Yaskawa INFORM job: R1_W39(90,0)R2.JBI

/JOB
//NAME R1_W39(90,0)R2
///FOLDERNAME KRIS-SCIANA
//POS
///NPOS 43,43,0,0,0,0
///TOOL 0
///POSTYPE PULSE
///PULSE
C00000=-48919,8763,-78145,-33912,86192,59629
C00001=-76192,74539,-3713,-7584,90498,58184
C00002=-85002,92103,26363,-6620,109146,2540
C00003=-82989,104273,47097,-9079,108858,2634
C00004=-80348,97044,37326,-14355,108478,2463
C00005=-80254,95353,36923,-14306,107890,2566
C00006=-81479,107840,53058,-15936,109964,1832
C00007=-88415,93116,33475,-16240,113040,-1015
C00008=-84401,99025,43999,-26670,113361,-1779
C00009=-80535,97927,39068,-19437,112108,13102
C00010=-80533,100008,38267,-19688,113585,12840
C00011=-95804,89991,27481,9151,105821,-39381
C00012=-93260,116784,65555,9230,104296,-50461
C00013=-88855,89918,29422,-607,100748,-50698
C00014=-93687,111856,59478,9313,105536,-50507
C00015=-89184,93974,34704,-472,103135,-51673
C00016=-95648,113896,64634,12639,107588,-50809
C00017=-91220,113921,60892,3414,106966,-50938
C00018=-94799,78029,20878,7231,106457,-51217
C00019=-94338,106165,52191,9314,107335,-50796
C00020=-97825,95185,41124,15323,107662,-50686
C00021=-97701,80312,23794,13413,106555,-50896
C00022=-97503,99676,37498,14313,114598,-56335
C00023=-97503,101438,37062,14468,115737,-56186
C00024=-130465,99741,46634,38839,105281,12352
C00025=-128682,100738,50844,38236,102897,12201
C00026=-125742,101757,54133,37646,100487,12538
C00027=-117769,55117,-4342,7008,90476,33925
C00028=-118319,57270,-3229,7217,90935,33791
C00029=-127381,86615,37635,37885,96810,10695
C00030=-119102,89171,33145,15718,101015,10229
C00031=-114648,83746,25609,1808,100380,9031
C00032=-114353,83732,25539,225,100330,11365
C00033=-114685,81630,17220,455,104304,11368
C00034=-111532,73347,14192,-9053,100688,13279
C00035=-111918,74812,15995,-7480,100020,12650
C00036=-113475,78376,20000,-2210,98733,12093
C00037=-114786,73408,9865,221,102241,12174
C00038=-116347,77074,8320,608,105082,11726
C00039=-119316,90665,15793,-710,107539,10303
C00040=-69963,31023,-55867,-11330,83895,10996
C00041=-61683,20403,-76764,12086,81991,2875
C00042=-8337,4565,-96754,54,101054,6652
BC00000=111077,708230,1070910
BC00001=111077,708230,1070910
BC00002=156085,702488,1070910
BC00003=156016,707290,1070907
BC00004=156002,708265,1070910
BC00005=156002,708265,1070910
BC00006=156016,707290,1070907
BC00007=156016,707290,1070907
BC00008=156016,707290,1070907
BC00009=133365,710613,1070910
BC00010=135484,706634,1070910
BC00011=156002,708265,1070910
BC00012=157117,904117,1084348
BC00013=156002,708265,1070904
BC00014=157117,904117,1084348
BC00015=156002,708265,1070904
BC00016=157117,904117,1084346
BC00017=156002,708265,1070904
BC00018=157117,904116,1084347
BC00019=156002,708265,1070904
BC00020=156002,708264,1070903
BC00021=156002,708263,1070903
BC00022=156002,708265,1070906
BC00023=156002,708265,1070906
BC00024=264527,676702,1070910
BC00025=264527,676702,1070910
BC00026=264527,676702,1070910
BC00027=264390,677222,1070910
BC00028=264390,677222,1070910
BC00029=264527,676702,1070910
BC00030=264527,676702,1070910
BC00031=264527,676702,1070910
BC00032=264527,676702,1070910
BC00033=264527,676702,1070910
BC00034=264528,676702,1070908
BC00035=264528,676702,1070907
BC00036=264528,676702,1070908
BC00037=264528,676702,1070908
BC00038=264528,676702,1070908
BC00039=264528,676702,1070908
BC00040=86198,708245,1070908
BC00041=129953,708245,1070908
BC00042=129953,672003,1070908
//INST
///DATE 2024/07/22 19:09
///ATTR SC,RW
///GROUP1 RB1,BS1
NOP
'r2_W39(90,0)
'Path S818
MOVJ C00000 BC00000 VJ=30.00
MOVJ C00001 BC00001 VJ=50.00
SFTOF
MOVJ C00002 BC00002 VJ=30.00
MOVL C00003 BC00003 V=100.0 PL=0
REFP 1 C00004 BC00004
REFP 2 C00005 BC00005
MACRO1 MJ#(0) ARGF7
ARCON
MOVL C00006 BC00006 V=10.0
MOVL C00007 BC00007 V=10.0
MOVL C00008 BC00008 V=10.0
ARCOF
MOVL C00009 BC00009 V=100.0
MOVL C00010 BC00010 V=100.0
SFTOF
'COMMENT
MOVL C00011 BC00011 V=100.0
COMM MOVL C00012 BC00012 V=100.0 PL=0  //OLD POSITION
MOVL C00013 BC00013 V=100.0 PL=0
MACRO1 MJ#(0) ARGF7
ARCON
COMM MOVL C00014 BC00014 V=10.0  //OLD POSITION
MOVL C00015 BC00015 V=10.0
COMM MOVL C00016 BC00016 V=10.0
MOVL C00017 BC00017 V=10.0
COMM MOVL C00018 BC00018 V=10.0  //OLD POSITION
MOVL C00019 BC00019 V=10.0
ARCON
MOVL C00020 BC00020 V=10.0
MOVL C00021 BC00021 V=10.0
ARCOF
SFTOF
MOVL C00022 BC00022 V=100.0
'W53
SFTOF
MOVJ C00023 BC00023 VJ=20.00
MOVJ C00024 BC00024 VJ=20.00
MOVL C00025 BC00025 V=83.3
MOVL C00026 BC00026 V=50.0
REFP 1 C00027 BC00027
REFP 2 C00028 BC00028
MACRO1 MJ#(0) ARGF7
ARCON
MOVL C00029 BC00029 V=8.3
MOVL C00030 BC00030 V=8.3
MOVL C00031 BC00031 V=8.3
MOVL C00032 BC00032 V=8.3
ARCOF
MOVL C00033 BC00033 V=83.3
MOVL C00034 BC00034 V=83.3
ARCON
MOVL C00035 BC00035 V=8.3
MOVL C00036 BC00036 V=8.3
ARCOF
MOVL C00037 BC00037 V=250.0
MOVJ C00038 BC00038 VJ=100.00
MOVJ C00039 BC00039 VJ=100.00
MOVJ C00040 BC00040 VJ=80.00
MOVJ C00041 BC00041 VJ=100.00
MOVJ C00042 BC00042 VJ=100.00
SFTOF
END
